{attribute 'conditionalshow'}
TYPE ST_ProfidriveParamSet :
	ARRAY[0..22] OF ST_ProfidriveParam; 
END_TYPE

(* stored: Version 1.1.0.1, ProductVersion 3.1.4024.12
   DUT ST_ProfidriveParamSet: Id {cf1cbdb5-41a7-0790-2d86-575d45bffa54} *)
